// TIA Portal project "S7anodownia3" (V15.1)

(* hardware
DEVICE "S7-1200 station_1"  S7-1200 Station
   slot 0: "Rack_0"  S7-1200 Rack  Rack  V1.0
   slot 1: "PLC 10.10.10.13"  CPU 1214C DC/DC/DC  6ES7 214-1AG40-0XB0  V4.3
DEVICE "GSD device_1"  GSD.Device.PN
   slot 0: "Rack"  Rack  V1.0
   slot 0: "smc-smc1"  JXCP1  JXCP1
      slot 0: "JXCP1"  JXCP1
      slot 1: "Interface"  Interface
         slot 1: "Port 1"  Port 1
         slot 2: "Port 2"  Port 2
      slot 1: "JXCP1_INPUT_1"  JXCP1_INPUT
         slot 0: "JXCP1_INPUT"  JXCP1_INPUT
      slot 2: "JXCP1_OUTPUT_1"  JXCP1_OUTPUT
         slot 0: "JXCP1_OUTPUT"  JXCP1_OUTPUT
*)

// ===== PLC "PLC 10.10.10.13"  CPU 1214C DC/DC/DC =====

VAR_GLOBAL   // PLC tag table "Default tag table"
   "System_Byte" AT %MB1 : Byte;
   "FirstScan" AT %M1.0 : Bool;
   "DiagStatusUpdate" AT %M1.1 : Bool;
   "AlwaysTRUE" AT %M1.2 : Bool;
   "AlwaysFALSE" AT %M1.3 : Bool;
   "Clock_Byte" AT %MB0 : Byte;
   "Clock_10Hz" AT %M0.0 : Bool;
   "Clock_5Hz" AT %M0.1 : Bool;
   "Clock_2.5Hz" AT %M0.2 : Bool;
   "Clock_2Hz" AT %M0.3 : Bool;
   "Clock_1.25Hz" AT %M0.4 : Bool;
   "Clock_1Hz" AT %M0.5 : Bool;
   "Clock_0.625Hz" AT %M0.6 : Bool;
   "Clock_0.5Hz" AT %M0.7 : Bool;
   "BTN W1 potwierdz zawieszke" AT %I0.0 : Bool;
   "LED W1 blokada zawieszki" AT %Q0.0 : Bool;
   "AUTO" AT %M50.0 : Bool;
   "A-EZ_dol" AT %Q0.1 : Bool;
   "A-EZ_gora" AT %Q0.2 : Bool;
   "tmp_wsadz" AT %M60.0 : Bool;
   "tmp_wyjmij" AT %M60.1 : Bool;
   "tmp_pobierz" AT %M60.2 : Bool;
END_VAR

VAR_GLOBAL   // PLC tag table "kroki"
   "A-krok_00" AT %M20.0 : Bool;   // Odczytanie kroku
   "A-krok_01" AT %M20.1 : Bool;   // rez
   "A-krok_02" AT %M20.2 : Bool;   // Przejazd dźwigu
   "A-krok_03" AT %M20.3 : Bool;   // rez
   "A-krok_04" AT %M20.4 : Bool;   // Operacja 1
   "A-krok_05" AT %M20.5 : Bool;   // rez
   "A-krok_06" AT %M20.6 : Bool;   // Operacja 2
   "A-krok_07" AT %M20.7 : Bool;   // rez
   "A-krok_08" AT %M21.0 : Bool;   // Usuniecie kroku z kolejki
   "A-krok_09" AT %M21.1 : Bool;   // rez
   "A-krok_99" AT %M22.1 : Bool;
   "A-krok_brak" AT %M22.2 : Bool;
   "A-krok_reset" AT %M22.3 : Bool;
   "A-krok_10" AT %M21.2 : Bool;   // Sprawdzenie zakonczenia
   "A-krok_11" AT %M21.3 : Bool;   // Ustawienie wanny 1
   "A-krok_12" AT %M21.4 : Bool;   // Przejazd dźwigu na wanne 1
END_VAR

TYPE "cParamKapiel"
   STRUCT
      tpraca : Int;
      tobciek : Int;
      tpowtorzenia : Int;
      tczas_pracy : Int;
      zakonczono : Bool;
      tukryj : Bool;
   END_STRUCT;
END_TYPE

TYPE "cProgram"
   STRUCT
      wanna : Int;
      offset : DTL;
      zawieszka : Int;
      operacja : String[10] := '          ';
      tpraca : Int;
      tobciek : Int;
      tpowtorzenia : Int;
   END_STRUCT;
END_TYPE

TYPE "cQueue"
   STRUCT
      maxSize : Int := 180;
      front : Int;
      rear : Int;
      count : Int;
      krok_count : Int;
      krok : Array[0..179] of "cProgram";
   END_STRUCT;
END_TYPE

// folder: SMC

TYPE "JXC_OUT"
VERSION : 0.1
   STRUCT
      OUT_0 : Bool;   // JXC Out 0
      OUT_1 : Bool;   // JXC Out 1
      OUT_2 : Bool;   // JXC Out 2
      OUT_3 : Bool;   // JXC Out 3
      OUT_4 : Bool;   // JXC Out 4
      OUT_5 : Bool;   // JXC Out 5
      Reserve1 : Bool;   // Reserve
      Reserve2 : Bool;   // Reserve
      BUSY : Bool;   // JXC -->PLC
      SVRE : Bool;   // JXC -->PLC
      SETON : Bool;   // JXC -->PLC
      INP : Bool;   // JXC -->PLC
      AREA : Bool;   // JXC -->PLC
      WAREA : Bool;   // JXC -->PLC
      ESTOP : Bool;   // JXC -->PLC
      ALARM : Bool;   // JXC -->PLC
      "Empty 1" : Bool;
      "Empty 2" : Bool;
      "Empty 3" : Bool;
      "Empty 4" : Bool;
      READY : Bool;
      "Empty 5" : Bool;
      "Empty 6" : Bool;
      "Empty 7" : Bool;
      "Empty 8" : Byte;
      CurrentPosition : DInt;   // Current position [0.01mm]
      CurrentSpeed : Int;   // Current speed [mm/s]
      CurrentForce : Int;   // Current force [%] {0..300}
      TargetPosition : DInt;   // Target position [0.01mm]
      ALARM1 : Byte;   // Alarm 1
      ALARM2 : Byte;   // Alarm 2
      ALARM3 : Byte;   // Alarm 3
      ALARM4 : Byte;   // Alarm 4
      "Empty 00" : DInt;   // Controller IF status Connect station
      "Empty 01" : DInt;   // Controller IF status Abnormal station
      "Empty 02" : DInt;   // Controller IF status reserve
      "Empty 03" : Byte;   // Controller IF status reserve
      "Empty 04" : Byte;
      "Empty 05" : Byte;
   END_STRUCT;
END_TYPE

TYPE "JXC_IN"
VERSION : 0.1
   STRUCT
      IN_0 : Bool;   // JXC IN 0
      IN_1 : Bool;   // JXC IN 1
      IN_2 : Bool;   // JXC IN 2
      IN_3 : Bool;   // JXC IN 3
      IN_4 : Bool;   // JXC IN 4
      IN_5 : Bool;   // JXC IN 5
      Reserve1 : Bool;   // Reserve
      Reserve2 : Bool;   // Reserve
      HOLD : Bool;   // PLC -> JXC
      SVON : Bool;   // PLC -> JXC
      DRIVE : Bool;   // PLC -> JXC
      RESET : Bool;   // PLC -> JXC
      SETUP : Bool;   // PLC -> JXC
      "JOG(-)" : Bool;   // PLC -> JXC
      "JOG(+)" : Bool;   // PLC -> JXC
      FLGTH : Bool;   // PLC -> JXC
      Reserve3 : Bool;   // PLC -> JXC
      SpeedRestriction : Bool;   // PLC -> JXC
      Reserve4 : Bool;   // PLC -> JXC
      Reserve5 : Bool;   // PLC -> JXC
      MovementMode : Bool;   // PLC -> JXC
      Speed_1 : Bool;   // PLC -> JXC
      Position_1 : Bool;   // PLC -> JXC
      Acceleration_1 : Bool;   // PLC -> JXC
      Deceleration_1 : Bool;   // PLC -> JXC
      PushingForce : Bool;   // PLC -> JXC
      TriggerLV : Bool;   // PLC -> JXC
      PushingSpeed : Bool;   // PLC -> JXC
      MovingForce : Bool;   // PLC -> JXC
      AreaOutput1 : Bool;   // PLC -> JXC
      AreaOutput2 : Bool;   // PLC -> JXC
      "In-PositionTolerRange" : Bool;   // PLC -> JXC
      StartFlag : Byte;   // PLC -> JXC
      MovementMode_1 : Byte;   // Reserve3
      SPEED : Int;   // Speed [mm/s]
      POSITION : DInt;   // Position [0.01mm]
      ACCELERATION : Int;   // Acceleration [mm/s^2]
      DECELERATION : Int;   // Deceleration [mm/s^2]
      PUSHING_FORCE : Int;   // Pushing force [10%] {0...30}
      TRIGGER_LV : Int;   // Trigger_LV [10%] {0...30}
      PUSHING_SPEED : Int;   // Pushing speed [mm/s]
      MOVING_FORCE : Int;   // Positioning thrust [10%] {0...30}
      AREA_1 : DInt;   // Area1
      AREA_2 : DInt;   // Area2
      InPOS_ToleranceRange : DInt;   // In position [0.01mm]
   END_STRUCT;
END_TYPE

TYPE "JXC"
   STRUCT
      in : Struct
         input_addr : Hw_Io;
         output_addr : Hw_Io;
         zalacz_naped : Bool;
         wybazuj : Bool;
         jog_skok : Bool;
         jog_plus : Bool;
         jog_minus : Bool;
         pozycja_mm : DInt;
         "predkosc_mm/s" : Int;
         start : Bool;
         reset : Bool;
      END_STRUCT;
      out : Struct
         zalaczony : Bool;
         wybazowany : Bool;
         w_bazie : Bool;
         busy : Bool;
         akt_pozycja : Real;
         akt_predkosc : Int;
         na_pozycji : Bool;
         error : Bool;
         error_nr : Int;
      END_STRUCT;
      params : Struct
         pozycja : Struct
            min : DInt := 0;
            max : DInt := 30000;
         END_STRUCT;
         predkosc : Struct
            min : Int := 6;
            max : Int := 50;
         END_STRUCT;
      END_STRUCT;
   END_STRUCT;
END_TYPE

// folder: TXRX

DATA_BLOCK "TXRX"   // DB1
{ S7_Optimized_Access := 'FALSE' }
VERSION : 0.1
   VAR
      cPlcParams : Struct
         actualTime : DTL;
         plc : Struct
            ready : Int;
         END_STRUCT;
      END_STRUCT;
   END_VAR
BEGIN
END_DATA_BLOCK

// folder: (top level)

ORGANIZATION_BLOCK "Main"   // OB1, LAD, ProgramCycle
TITLE = "Main Program Sweep (Cycle)"
{ S7_Optimized_Access := 'TRUE' }
VERSION : 0.1
   VAR_INPUT
      Initial_Call : Bool;   // Initial call of this OB
      Remanence : Bool;   // =True, if remanent data are available
   END_VAR
   VAR_TEMP
      aa : DInt;
      bb : DTL;
   END_VAR
BEGIN

REGION Network 1: Komunikacja z PLC
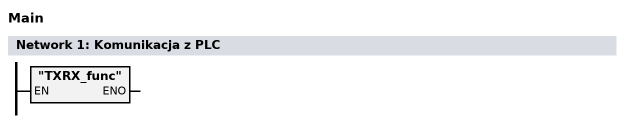
   RUNG wire#powerrail
      "TXRX_func"()
   END_RUNG
   // the same network as SCL:
   "TXRX_func"();
END_REGION
END_ORGANIZATION_BLOCK

// folder: TXRX

FUNCTION "TXRX_func" : Void   // FC1, LAD
{ S7_Optimized_Access := 'TRUE' }
VERSION : 0.1
   VAR_TEMP
      TXRXrel_val : Int;
   END_VAR
BEGIN

REGION Network 1: Odczyt aktualnego czasu
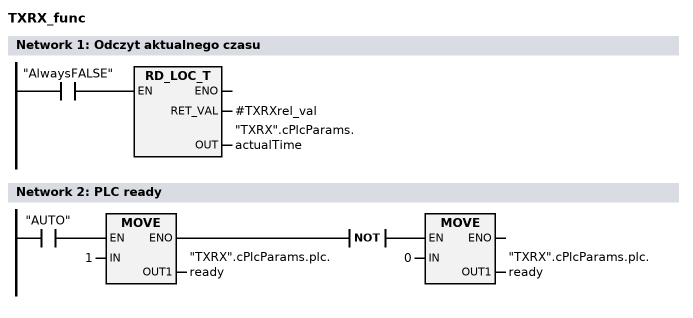
   IF "AlwaysFALSE" THEN #TXRXrel_val := RD_LOC_T(OUT => "TXRX".cPlcParams.actualTime); END_IF;
END_REGION

REGION Network 2: PLC ready
   RUNG wire#powerrail
      Contact( "AUTO" )
      Move(in := 1, out1 => "TXRX".cPlcParams.plc.ready)
      Not()
      Move(in := 0, out1 => "TXRX".cPlcParams.plc.ready)
   END_RUNG
   // the same network as SCL:
   IF "AUTO" THEN "TXRX".cPlcParams.plc.ready := 1; END_IF;
   IF NOT "AUTO" THEN "TXRX".cPlcParams.plc.ready := 0; END_IF;
END_REGION
END_FUNCTION